{attribute 'linkalways'}
{attribute 'no_explicit_call' := 'This FB is a CLASS and must be accessed using methods or properties'}
{attribute 'enable_dynamic_creation'}
FUNCTION_BLOCK _ETcVnSalientFeaturesMethod EXTENDS EnumDatatypeBase
VAR
	localData : ETcVnSalientFeaturesMethod;
	activeData : REFERENCE TO ETcVnSalientFeaturesMethod;
	enumBaseDatatype : _UDINT(localData);
END_VAR

METHOD PRIVATE AddLocalEnumeration
VAR_INPUT
	Enumeration : T_MAXSTRING;
	Value : ETcVnSalientFeaturesMethod;
END_VAR
AddEnumeration(Enumeration, Value);
END_METHOD

PROPERTY PUBLIC Address : PVOID
GET
Address := ADR(activeData);
END_GET
END_PROPERTY

METHOD PUBLIC ClearReference
VAR_INPUT
END_VAR
activeData REF= localData;
SetBaseDatatypeReference();
END_METHOD

METHOD PUBLIC Clone : I_Datatype
VAR
    pClone : POINTER TO _ETcVnSalientFeaturesMethod;
END_VAR
pClone := __NEW(_ETcVnSalientFeaturesMethod(InitialValue := Value));
IF pClone = 0 THEN
    RETURN;
END_IF
Clone := pClone^;
END_METHOD

METHOD FB_init : BOOL
VAR_INPUT
	bInitRetains : BOOL; // if TRUE, the retain variables are initialized (warm start / cold start)
	bInCopyCode : BOOL;  // if TRUE, the instance afterwards gets moved into the copy code (online change)
	InitialValue : ETcVnSalientFeaturesMethod;
END_VAR
localData := InitialValue;
AddBaseDatatype(enumBaseDatatype);
ClearReference();

AddLocalEnumeration('TCVN_SFM_WALSH_CODE', ETcVnSalientFeaturesMethod.TCVN_SFM_WALSH_CODE);
AddLocalEnumeration('TCVN_SFM_SOBEL', ETcVnSalientFeaturesMethod.TCVN_SFM_SOBEL);
END_METHOD

PROPERTY PUBLIC Identifier : T_MAXSTRING
GET
Identifier := 'ETcVnSalientFeaturesMethod';
END_GET
END_PROPERTY

METHOD IsEnumeratorValueEqual : BOOL
VAR_INPUT
	Enumerator : I_KeyValueForwardEnumerator;
END_VAR
VAR
	storedValue : ETcVnSalientFeaturesMethod;
END_VAR
IF NOT Enumerator.TryGet(storedValue) THEN
	RETURN;
END_IF

IsEnumeratorValueEqual := storedValue = activeData;
END_METHOD

METHOD PUBLIC MakeReferenceTo
VAR_INPUT
	ReferenceTarget : REFERENCE TO ETcVnSalientFeaturesMethod;
END_VAR
activeData REF= ReferenceTarget;
SetBaseDatatypeReference();
END_METHOD

METHOD PROTECTED SetBaseDatatypeReference
VAR_INPUT
END_VAR
enumBaseDatatype.MakeReferenceTo(activeData);
END_METHOD

PROPERTY PUBLIC Size : UDINT
GET
Size := SIZEOF(activeData);
END_GET
END_PROPERTY

METHOD TryMakeReferenceTo : BOOL
VAR_INPUT
	Target : I_Datatype;
END_VAR
VAR
	pTargetData : POINTER TO ETcVnSalientFeaturesMethod;
END_VAR
IF NOT IsEquivalentTo(Target) THEN
	RETURN;
END_IF

pTargetData := Target.Address;
activeData REF= pTargetData^;
SetBaseDatatypeReference();
TryMakeReferenceTo := TRUE;
END_METHOD

PROPERTY PUBLIC Value : ETcVnSalientFeaturesMethod
GET
Value := activeData;
END_GET
SET
activeData := Value;
END_SET
END_PROPERTY

END_FUNCTION_BLOCK

(* stored: Version 1.1.0.1, ProductVersion 3.1.4026.13
   POU _ETcVnSalientFeaturesMethod: Id {ba06b2ea-2ef4-4e29-b7b8-7370c19065b7}, SpecialFunc None
   Folder Core: Id {3ce9f64b-7e9b-49dd-96b3-4ea92aa3e233}
   Folder Protected: Id {7456e1c2-6e8d-475d-ba64-3051fd8cf17d}
   Folder Customize: Id {366fbad4-35fb-4e0d-889f-5bc1fcea0f7b}
   Folder Constructor: Id {16019516-c510-4aee-9f4a-1cfd18de1a68}
   Folder Private: Id {0562efa3-cf19-4de5-88e8-c82753f3b231}
   Folder Protected: Id {18e4d330-e97b-4efa-8b28-9ceabbb71db2}
   Method AddLocalEnumeration: Id {7ee6d82c-91a4-4b33-a536-c1c33207af03}
   Property Address: Id {59440a52-02a6-4e8d-bc40-08169e4f3019}
   Get Get: Id {8a05dfe8-96a0-46bc-97eb-22024e7d9556}
   Method ClearReference: Id {a2994203-df38-4f29-95d5-69ae76fe7e13}
   Method Clone: Id {5200c43c-47cb-45ab-809e-25fdff3308e2}
   Method FB_init: Id {c1fe99ab-4249-4205-9e35-eea174af6c48}
   Property Identifier: Id {e01cc974-7851-487d-bafb-a08ae2b5a757}
   Get Get: Id {667a709a-1123-444b-8762-f0de9d5f6910}
   Method IsEnumeratorValueEqual: Id {5c5278cf-bd69-4fdb-ab07-62389f19779c}
   Method MakeReferenceTo: Id {7e8c6a32-21e7-42fb-981a-bb0e0eb9ca3b}
   Method SetBaseDatatypeReference: Id {0d8e7a70-66b8-4534-aa6f-9e52cbce80a5}
   Property Size: Id {1bfe6a6c-7867-43d7-b3f4-99ff5123bdbf}
   Get Get: Id {0415ee55-89dd-4a14-bcb7-024322d63f82}
   Method TryMakeReferenceTo: Id {14e7007d-d860-45b4-b8f1-ea305b9649b9}
   Property Value: Id {c47923d5-0efd-40e5-9ded-9c46c0318d92}
   Get Get: Id {5a72b536-ff4e-43d6-9065-4473f34619df}
   Set Set: Id {aa90a05a-846c-45fe-937e-54fc93558b14} *)
